FUNCTION_BLOCK FB_Ampel
VAR_INPUT
	eState : eBetriebszustand;
END_VAR
VAR_OUTPUT
	bAmpelGrun : BOOL;
	bAmpelRot : BOOL;
	bAmpelGelb : BOOL;
END_VAR
VAR
	fbBlinklicht : FB_Blinklicht;
END_VAR

CASE eState OF
	eBetriebszustand.Off:
		bAmpelGrun := FALSE;
		bAmpelGelb := FALSE;
		bAmpelRot := TRUE;
	
	eBetriebszustand.Error:
		bAmpelGrun := FALSE;
		bAmpelGelb := FALSE;
		fbBlinklicht(bStartStop:= TRUE, tPeriode:= T#1S, bBlink=> bAmpelRot );
	
	eBetriebszustand.Setup:
		bAmpelGrun := FALSE;
		bAmpelGelb := TRUE;
		bAmpelRot := FALSE;
	
	eBetriebszustand.Warning:
		bAmpelGrun := FALSE;
		fbBlinklicht(bStartStop:= TRUE, tPeriode:= T#1S, bBlink=> bAmpelGelb );
		bAmpelRot := FALSE;
		
	eBetriebszustand.Init:
		bAmpelGrun := TRUE;
		bAmpelGelb := TRUE;
		bAmpelRot := FALSE;
	
	eBetriebszustand.Ready:
		bAmpelGrun := TRUE;
		bAmpelGelb := FALSE;
		bAmpelRot := FALSE;
	
	eBetriebszustand.Production:
		bAmpelRot := FALSE;
		fbBlinklicht(bStartStop:= TRUE , tPeriode:= T#1S, bBlink=> bAmpelGrun);
		fbBlinklicht(bStartStop:= TRUE , tPeriode:= T#1S, bBlink=> bAmpelGelb);
	
	eBetriebszustand.Done:
		fbBlinklicht(bStartStop:= TRUE , tPeriode:= T#1S, bBlink=> bAmpelGrun);
		bAmpelGelb := FALSE;
		bAmpelRot := FALSE;
		
	eBetriebszustand.Stop:
		bAmpelGrun := FALSE;
		fbBlinklicht(bStartStop:= TRUE , tPeriode:= T#1S, bBlink=> bAmpelRot);
		fbBlinklicht(bStartStop:= TRUE , tPeriode:= T#1S, bBlink=> bAmpelGelb);
	
	
	
	
	
	
	
END_CASE

END_FUNCTION_BLOCK

(* stored: Version 1.1.0.1, ProductVersion 3.1.4024.15
   POU FB_Ampel: Id {366d4720-12a4-4ad2-980d-adb7cd3a227b}, SpecialFunc None *)
